TYPE TcoControlledZone_Status :
STRUCT
	ActionDescription : STRING(100);	
	State : TcoControledZone_Info;	
	
END_STRUCT
END_TYPE

(* stored: Version 1.1.0.1
   DUT TcoControlledZone_Status: Id {ca7d523b-825d-4e92-8f2b-06548eab290f} *)
